// TIA Portal V17 export
// export: Created 2021-12-03T08:13:12.5470958Z, ExportSetting WithDefaults, DisplayName Totally Integrated Automation Portal, DisplayVersion V17, DisplayName TIA Portal Openness, DisplayVersion V17, DisplayName TIA Portal Version Control Interface, DisplayVersion V17, DisplayName STEP 7 Professional, DisplayVersion V17, DisplayName STEP 7 Safety, DisplayVersion V17, DisplayName WinCC Advanced, DisplayVersion V17
DATA_BLOCK "FDBI_TmSelChillOn"   // DB706, F_DB
VERSION : 0.1
// stored: AutoNumber false, InstanceOfName FFB_TmSel, InstanceOfType FB
"FFB_TmSel"
   // VAR_INPUT
   //    I_Sel_2 : Bool;
   //    I_Time_1 : Time;
   //    I_Time_2 : Time;
   // END_VAR
   // VAR_OUTPUT
   //    O_Sel_2 : Bool;
   //    O_SelTime : Time;
   // END_VAR
BEGIN
END_DATA_BLOCK
